PROGRAM _05_Config_Drain
VAR
v015_Grv :fValve;
v016_Grv2 :fValve;
v017_Pump :fValve;
s018_LvlHT :dutpul;
s019_TempHT :fTemp;
v020_HT :fValve;
v021_WaterHT :fValve;
END_VAR

(*-------------------------------------------------------------------------------------------------------*)
(*-------------------------------------------------------------------------------------------------------*)

(*------------------------------------------------------------------------------------------------------*)
(*Comprobar si hay sensor de nivel del Vaciado HT *)
Mc._05_DRAIN.xLvlHT		:=Mc._05_DRAIN.s018_LvlHT.xPul;


(*Comprobar si hay PT100 del vaciado HT *)
Mc._05_DRAIN.iTempHT	:= REAL_TO_INT (Mc._05_DRAIN.s019_TempHT.rValue);



//v015_Gvr
v015_Grv(valv:=mc._05_DRAIN.v015_Grv );

//v016_Grv2
v016_Grv2 (valv:= mc._05_DRAIN.v016_Grv2);

//v017_Pump
v017_Pump(valv:=mc._05_DRAIN.v017_Pump);

//s018_LvlHT
s018_LvlHT:=mc._05_DRAIN.s018_LvlHT;
(*
//s019_TempHT 
s019_TempHT.Temp.rAna_min:=0;
s019_TempHT.Temp.rAna_max:=1500;
s019_TempHT.Temp.rUf_min:=0;
s019_TempHT.Temp.rUf_max:=150;
//s019_TempHT.Temp.
*)
//v020_HT
v020_HT(valv:=mc._05_DRAIN.v020_HT);

//v021_WaterHT
v021_WaterHT (valv:=mc._05_DRAIN.v021_WaterHT);

END_PROGRAM

(* stored: Version 1.1.0.1, ProductVersion 3.1.4024.10
   POU _05_Config_Drain: Id {49f13463-3f0a-4bbd-a176-e4e9f3f8da21}, SpecialFunc None *)
